// Mitsubishi GX Works2 project: TEST   PLC: FX2N/FX2NC

PROGRAM MAIN
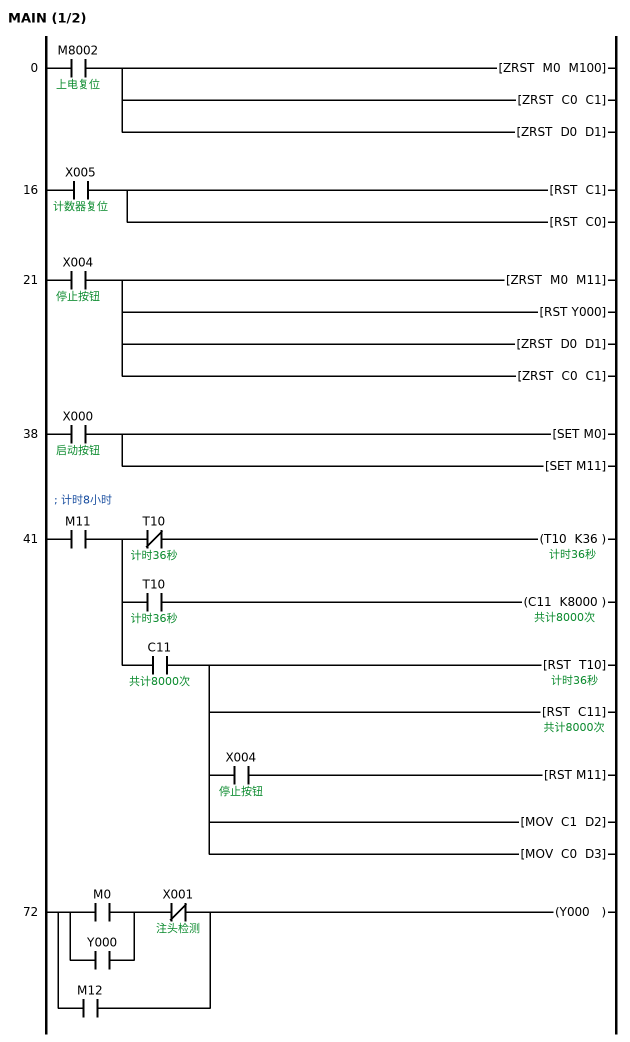
0     LD      M8002  ; 上电复位
      ZRST    M0 M100
      ZRST    C0 C1
      ZRST    D0 D1
16    LD      X005  ; 计数器复位
      RST     C1
      RST     C0
21    LD      X004  ; 停止按钮
      ZRST    M0 M11
      RST     Y000
      ZRST    D0 D1
      ZRST    C0 C1
38    LD      X000  ; 启动按钮
      SET     M0
      SET     M11
; 计时8小时
41    LD      M11
      MPS
      ANI     T10  ; 计时36秒
      OUT     T10 K36  ; 计时36秒
      MRD
      AND     T10  ; 计时36秒
      OUT     C11 K8000  ; 共计8000次
      MPP
      AND     C11  ; 共计8000次
      RST     T10  ; 计时36秒
      RST     C11  ; 共计8000次
      MPS
      AND     X004  ; 停止按钮
      RST     M11
      MPP
      MOV     C1 D2
      MOV     C0 D3
72    LD      M0
      OR      Y000
      ANI     X001  ; 注头检测
      OR      M12
      OUT     Y000
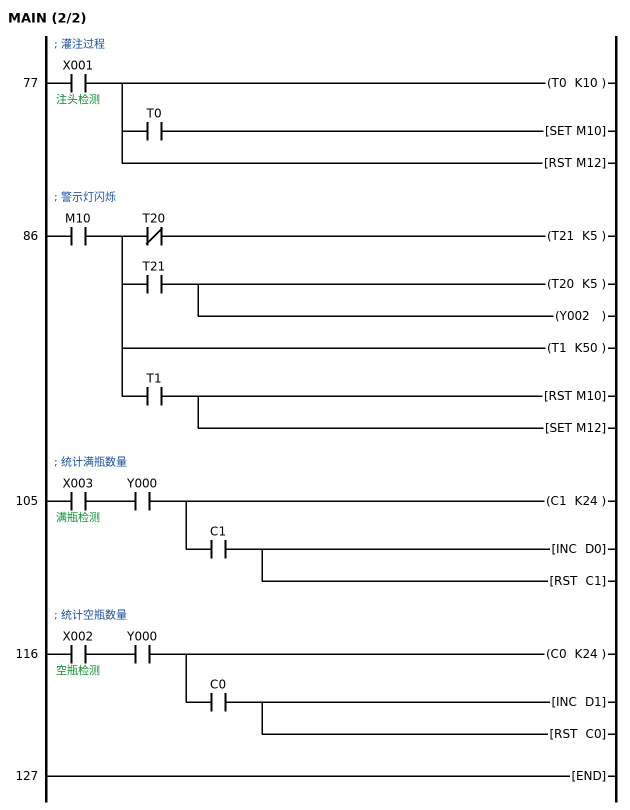
; 灌注过程
77    LD      X001  ; 注头检测
      OUT     T0 K10
      MPS
      AND     T0
      SET     M10
      MPP
      RST     M12
; 警示灯闪烁
86    LD      M10
      MPS
      ANI     T20
      OUT     T21 K5
      MRD
      AND     T21
      OUT     T20 K5
      OUT     Y002
      MPP
      OUT     T1 K50
      AND     T1
      RST     M10
      SET     M12
; 统计满瓶数量
105   LD      X003  ; 满瓶检测
      AND     Y000
      OUT     C1 K24
      AND     C1
      INC     D0
      RST     C1
; 统计空瓶数量
116   LD      X002  ; 空瓶检测
      AND     Y000
      OUT     C0 K24
      AND     C0
      INC     D1
      RST     C0
127   END
END_PROGRAM
